//{{V2}}
DATA_BLOCK DB10

AUTHOR:mh
FAMILY:nb
NAME:nb
VERSION:1.0


       STRUCT
         b0:INT
         b1:INT
         b2:INT
         b3:INT
         b4:INT
         b5:INT
         b6:INT
         b7:INT
         b8:INT
         b9:INT
       END_STRUCT
BEGIN

       b0:=6
       b1:=1
       b2:=9
       b3:=10
       b4:=4
       b5:=2
       b6:=10
       b7:=103
       b8:=23
       b9:=10
END_DATA_BLOCK
